ABB RobotStudio station: Lab1.2.rsstn

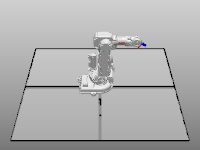
Station Lab1.2 (saved by RobotStudio 21.2.9526.0)
Controller IRB140
  mechanical unit ROB_1: IRB140_6_81_C_03_3, 6 joints, base frame (0, 0, 0) mm
Layout (positions relative to the parent item):
  - IRB140_6_81_C_03_3 [mechanism, from Robots\IRB140_6_81_C_G_03.rslib] at (0, 0, 0) mm; joint values [0, 0, 0, 0, 0.5236, 0] (rad or m)
